SUBAPPLICATION Uebung_012c_AX (* Numeric Value Input und Speichern INI mit Subapp *)
  (* Standard: 61499-2; Description: Copyright (c) 2023 Meisterschulen am Ostbahnhof This program and the accompanying materials are made available under the terms of the Eclipse Public License 2.0 which is available at https://www.eclipse.org/legal/epl-2.0/ SPDX-License-Identifier: EPL-2.0 *)
  (* Version 1.0, 2023-10-23, Franz Höpfinger, Meisterschulen am Ostbahnhof, initial API and implementation and/or initial documentation *)
  PACKAGE Uebungen;
  IMPORT Uebungen::const::NVS::NVS_Keys::KEY_I1_STORE;
  IMPORT Uebungen::const::NVS::NVS_Keys::SECTION_I1_STORE;
  IMPORT Uebungen::const::UT::DefaultPool::InputNumber_I1;
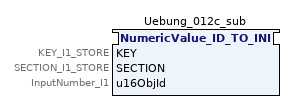
  SUBAPPS
    Uebung_012c_sub : MyLib::sys::NumericValue_ID_TO_INI(KEY := KEY_I1_STORE, SECTION := SECTION_I1_STORE, u16ObjId := InputNumber_I1);
  END_SUBAPPS
END_SUBAPPLICATION
